FUNCTION_BLOCK EM_Doors EXTENDS EM_Base
VAR CONSTANT 
	c_nResultDataSize : UINT := 20;
END_VAR
VAR
//------------------------------------------//
//Control Modules (Devices)
	s_cmSpeedDoorOuter : CM_SpeedDoor;
	s_cmDoorLockCleanroom : CM_DoorLock;
//------------------------------------------//

//------------------------------------------//
//Inputs
	s_diTableDownSensor	: FB_DigInput;
	s_diBtnTableDown	: FB_DigInput;
	s_diBtnStop			: FB_DigInput;
	
//------------------------------------------//
	s_doRelayTableDown : FB_DigOutput;
//------------------------------------------//
//Outputs

//------------------------------------------//

//------------------------------------------//
//Params
	//Tool settings
	s_fbParamToolHardwareNr				: FB_HmiParamHandler;
    s_fbParamToolSoftwareVersion		: FB_HmiParamHandler;

	s_fbParamName						: FB_HmiParamHandler;
	s_fbParamNumber						: FB_HmiParamHandler;
	s_fbParamRevision                   : FB_HmiParamHandler;
	
	s_fbParamTeslaMeterIp				: FB_HmiParamHandler;
	s_fbParamTeslaMeterPort				: FB_HmiParamHandler;
	
	//Product settings (Maybe)
	s_fbParamTotalStroke				: FB_HmiParamHandler;
	s_fbParamStepStroke					: FB_HmiParamHandler;
	s_fbParamAveragingNumberTest		: FB_HmiParamHandler;
	
	s_fbParamaMaxMagnitudeCriteria		: FB_HmiParamHandler;
	
	s_fbParamRefIduBottom				: FB_HmiParamHandler;
	s_fbParamRefItm                     : FB_HmiParamHandler;
	s_fbParamRefCenterTpmPipe           : FB_HmiParamHandler;
	s_fbParamRefCpValve					: FB_HmiParamHandler;
//------------------------------------------//

//------------------------------------------//
//Variables
	s_sTestResult 						: STRING;
	
	s_eCurrentTest						: E_TestMode;
	s_stCommandsTesla					: ST_SCPI_TeslaCommands;
//------------------------------------------//

//------------------------------------------//
//Sensor data	
	s_aMagneticX						: ARRAY[0..c_nResultDataSize] OF LREAL;
	s_aMagneticY						: ARRAY[0..c_nResultDataSize] OF LREAL;
	s_aMagneticZ						: ARRAY[0..c_nResultDataSize] OF LREAL;
	s_aMagneticMagnitude				: ARRAY[0..c_nResultDataSize] OF LREAL;
	s_aProbePositionZ					: ARRAY[0..c_nResultDataSize] OF LREAL;
	
	s_sXMLData							: STRING(Param_Project.n_MaxLenghtXmlDbRow*Param_Project.n_NumberofRowsXmlDb);
	
	s_aHmi_MagneticTest					: ARRAY[1..3,0..c_nResultDataSize] OF ST_POINT;
	
//	s_aHmi_ProbePositionZ				: ARRAY[1..1,1..GVL_Datalogging.c_nHmiLogSize] OF ST_POINT;
//------------------------------------------//

//------------------------------------------//
//Alarms

//------------------------------------------//

//------------------------------------------//
//Hmi
	s_nToHmiStepNr						: INT;
	s_nToHmiMaxStepNr					: INT;
	s_sToHmiInstructionText				: T_MAXSTRING;
	s_sToHmiProcedure					: T_MAXSTRING;
	
	s_fbHmiBtnStart						: FB_HmiBtn;
	s_fbHmiBtnStop						: FB_HmiBtn;	
	s_fbHmiBtnDiagnosticsLogging		: FB_HmiBtn;
	
	s_fbHmiProbeMotor 					: Hmi_Motor_Base;
	
	s_fbHmiBtnEnableMotor				: FB_HmiBtn;
	s_fbHmiBtnHomeMotor					: FB_HmiBtn;
	s_fbHmiBtnGetField					: FB_HmiBtn;
	
	s_fbHmiLedHomedMotor				: FB_HmiLed;
	s_fbHmiTableDownPressed				: FB_HmiLed;
	s_fbHmiStopPressed					: FB_HmiLed;
	s_fbHmiTableDownSensor				: FB_HmiLed;
//------------------------------------------//
END_VAR


SUPER^();

METHOD Protected _m_Alarms : BOOL
IF NOT SUPER^._m_Alarms() THEN
	RETURN;
END_IF

_m_Alarms := TRUE;
END_METHOD

METHOD PRIVATE _m_DatabaseMagnetic : BOOL
VAR_INPUT
	i_bCmdReset						: BOOL;
	i_sPassFail						: STRING;
END_VAR
VAR_INST
	s_aDbColumns				: ARRAY[1..GVL_DataLogging.c_nDbColumnMagnetic] OF STRING;
	s_aDbColumnValues			: ARRAY[1..GVL_DataLogging.c_nDbColumnMagnetic] OF STRING;
	
	s_nCounterDbLogging				: UINT := 1;
END_VAR
IF i_bCmdReset THEN
	s_nCounterDbLogging 	:= 1;
	
	MEMSET(ADR(s_aDbColumns), 0 , SIZEOF(s_aDbColumns));
	MEMSET(ADR(s_aDbColumnValues), 0 , SIZEOF(s_aDbColumnValues));	

	s_aDbColumns[1] 		:= 'TestTool Hardware Nr';
	s_aDbColumns[2] 		:= 'TestTool Software Version';
	s_aDbColumns[3] 		:= 'User';
	s_aDbColumns[4] 		:= 'Serial number';
	s_aDbColumns[5] 		:= '12NC';
	s_aDbColumns[6] 		:= 'Notes';
	s_aDbColumns[7] 		:= 'PassFail';
	s_aDbColumns[8] 		:= 'Message';
	s_aDbColumns[9] 		:= 'Measurement';
	
	s_aDbColumnValues[1] 	:= GVL_DataLogging.g_stReportData.CabinetSerialNumber;
	s_aDbColumnValues[2] 	:= GVL_DataLogging.g_stReportData.TesterSoftwareVersion;
	s_aDbColumnValues[3] 	:= GVL.g_sUser;
	s_aDbColumnValues[4] 	:= GVL_DataLogging.g_stReportData.SerialNumber;;
	s_aDbColumnValues[5] 	:= CONCAT(s_fbParamNumber.p_sValue, CONCAT('^' ,TO_STRING(TO_INT(s_fbParamRevision.p_fValue))));
	s_aDbColumnValues[6] 	:= GVL.g_sNotesEntry;
	s_aDbColumnValues[7]  	:= i_sPassFail;
		
	IF GVL_KMWEGenericLib.g_fbAlarmManager.p_bAlarmActive THEN
		s_aDbColumnValues[8] 	:= 'Stopped due to Alarm';
	ELSE
		s_aDbColumnValues[8] 	:= '';
	END_IF
	
END_IF

IF s_nCounterDbLogging < GVL_DataLogging.c_nDbColumnMagnetic THEN
	IF GVL_Datalogging.g_fbSqlDatabase.m_UpdateTableValue(i_sTableName					:= GVL_DataLogging.c_sTableNameMagnetic,
															i_sIdentificationColumnName := GVL_DataLogging.c_sIdentificationColumnDataTime,
															i_sIdentificationValue		:= GVL_KMWEGenericLib.g_fbCurrentTime.p_sCurrentDateTime_DB, 
															i_sColumnName				:= s_aDbColumns[s_nCounterDbLogging], 
															i_sColumnValue				:= s_aDbColumnValues[s_nCounterDbLogging])
	THEN
		IF s_nCounterDbLogging <=  GVL_DataLogging.c_nDbColumnMagnetic THEN
			s_nCounterDbLogging := s_nCounterDbLogging + 1;
		END_IF
	END_IF
ELSIF s_nCounterDbLogging = GVL_DataLogging.c_nDbColumnMagnetic THEN
	IF GVL_Datalogging.g_fbSqlDatabase.m_UpdateTableXml(i_sTableName					:= GVL_DataLogging.c_sTableNameMagnetic,
															i_sIdentificationColumnName := GVL_DataLogging.c_sIdentificationColumnDataTime,
															i_sIdentificationValue		:= GVL_KMWEGenericLib.g_fbCurrentTime.p_sCurrentDateTime_DB, 
															i_sColumnName				:= s_aDbColumns[s_nCounterDbLogging], 
															i_addrColumnValue			:= ADR(s_sXMLData))
	THEN
		IF s_nCounterDbLogging <=  GVL_DataLogging.c_nDbColumnMagnetic THEN
			s_nCounterDbLogging := s_nCounterDbLogging + 1;
		END_IF
	END_IF
END_IF

_m_DatabaseMagnetic := s_nCounterDbLogging > GVL_DataLogging.c_nDbColumnMagnetic;
END_METHOD

METHOD Protected _m_Devices : BOOL
VAR_INPUT
END_VAR
IF NOT SUPER^._m_Devices() THEN
	RETURN;
END_IF

s_CmProbeMotor(
	i_bReqEnable					:= , //written in test procedure or manual 
	i_eCtrlMode						:= i_eCtrlMode, 
	i_bCmdReset						:= i_bCmdReset, 
	i_sCmName						:= 'Probe motor');	
	
s_CmTeslaMeter(
	i_bReqEnable					:= , //written in test procedure or manual  
	i_eCtrlMode						:= i_eCtrlMode, 
	i_bCmdReset						:= i_bCmdReset, 
	i_sCmName						:= 'Tesla meter');
	
_m_Devices := TRUE;
END_METHOD

METHOD PRIVATE _m_GetMagneticField : E_STATE
VAR_INPUT
	i_bCmdReset			: BOOL;
END_VAR
VAR_OUTPUT
	q_fMagneticX		: LREAL;
	q_fMagneticY		: LREAL;
	q_fMagneticZ		: LREAL;
END_VAR
VAR_INST
	//Sequence control
	s_eSequence				: E_ModuleSeqBase;
	s_fbSeqControl			: FB_SeqControl;
	
	s_nInternalStep			: UINT := 0;
	
	//Communication
	s_aReplyBuffer			: ARRAY[1..100] OF T_MAXSTRING; //Tesla
	s_aResults				: ARRAY[1..10 ] OF T_MAXSTRING;	//Tesla
	s_sReply				: T_MAXSTRING;
	s_nIndexReply 			: UDINT := 1;
	s_nIndexResults			: UDINT := 1;
	
	t_nMeasurementsReceived		: UDINT := 1;

	//Measurements
	s_aMagneticXAve			: ARRAY[1..100] OF LREAL;
	s_aMagneticYAve			: ARRAY[1..100] OF LREAL;
	s_aMagneticZAve			: ARRAY[1..100] OF LREAL;
END_VAR
VAR
	t_nCyclceReplies			: UDINT := 1;
	
	t_fAveragingX				: LREAL;
	t_fAveragingY				: LREAL;
	t_fAveragingZ				: LREAL;

END_VAR
s_fbSeqControl(
	i_nSeqStep:= s_eSequence, 
	i_sStepName:= TO_STRING(s_eSequence), 
	i_bCmdReset:= i_bCmdReset, 
	i_bStaError:= FALSE,  
	q_eActState=> _m_GetMagneticField);
	
CASE s_eSequence OF
	E_ModuleSeqBase.Idle:
		;
		
	E_ModuleSeqBase.Start:
		IF s_fbSeqControl.q_bStaEntry THEN
			s_nInternalStep := s_nInternalStep + 1;
		END_IF
		
		IF s_fbSeqControl.q_tmStepTime > T#2S OR s_nInternalStep > 1 THEN
			IF s_CmTeslaMeter.m_SendCommand(i_sCommand := s_stCommandsTesla.sGetMeasurents , i_bAddCRChar := TRUE) THEN
				s_eSequence 	:= E_ModuleSeqBase.Busy;
			END_IF
		END_IF

	E_ModuleSeqBase.Busy:
		IF s_fbSeqControl.q_bStaEntry THEN
			t_nMeasurementsReceived := 1;
		END_IF
		
		s_CmTeslaMeter.m_ReadReplyBuffer(q_sReply => s_sReply);
			
		IF s_sReply <> 'No reply' THEN
			IF t_nMeasurementsReceived = 1 THEN
				s_aReplyBuffer[t_nCyclceReplies] := '';
				t_nMeasurementsReceived := 2;
			ELSIF t_nMeasurementsReceived = 2 THEN
				s_aMagneticXAve[s_nInternalStep] := TO_LREAL(s_aReplyBuffer[t_nCyclceReplies]);
				s_aMagneticXAve[s_nInternalStep] := TO_LREAL(s_sReply);
				s_aReplyBuffer[t_nCyclceReplies] := '';
				t_nMeasurementsReceived := 3;
			ELSIF t_nMeasurementsReceived = 3 THEN
				s_aMagneticYAve[s_nInternalStep] := TO_LREAL(s_aReplyBuffer[t_nCyclceReplies]);
				s_aMagneticYAve[s_nInternalStep] := TO_LREAL(s_sReply);
				s_aReplyBuffer[t_nCyclceReplies] := '';
				t_nMeasurementsReceived := 4;
			ELSIF t_nMeasurementsReceived = 4 THEN
				s_aMagneticZAve[s_nInternalStep] := TO_LREAL(s_aReplyBuffer[t_nCyclceReplies]);
				s_aMagneticZAve[s_nInternalStep] := TO_LREAL(s_sReply);
				s_aReplyBuffer[t_nCyclceReplies] := '';

				IF s_nInternalStep = TO_UINT(s_fbParamAveragingNumberTest.p_fValue) THEN
					s_eSequence := E_ModuleSeqBase.Ready;
				ELSE
					s_eSequence := E_ModuleSeqBase.Start;
				END_IF 
			END_IF
		END_IF

	E_ModuleSeqBase.Ready:
		IF s_fbSeqControl.q_bStaEntry THEN
			s_nInternalStep := 0;
			
			t_fAveragingX	:= 0;
			t_fAveragingY	:= 0;
			t_fAveragingZ	:= 0;
 
			MEMSET(ADR(s_aReplyBuffer)			, 0, SIZEOF(s_aReplyBuffer));
			MEMSET(ADR(s_aResults)				, 0, SIZEOF(s_aResults));
		END_IF
		
		FOR t_nCyclceReplies := 1 TO 100 DO
			t_fAveragingX := t_fAveragingX + s_aMagneticXAve[t_nCyclceReplies];
			t_fAveragingY := t_fAveragingY + s_aMagneticYAve[t_nCyclceReplies];
			t_fAveragingZ := t_fAveragingZ + s_aMagneticZAve[t_nCyclceReplies];

			IF t_nCyclceReplies = 100 THEN
			MEMSET(ADR(s_aMagneticXAve)			, 0, SIZEOF(s_aMagneticXAve));
			MEMSET(ADR(s_aMagneticYAve)			, 0, SIZEOF(s_aMagneticYAve));
			MEMSET(ADR(s_aMagneticZAve)			, 0, SIZEOF(s_aMagneticZAve));				
			END_IF
		END_FOR
			
			q_fMagneticX	:= t_fAveragingX/s_fbParamAveragingNumberTest.p_fValue;
			q_fMagneticY	:= t_fAveragingY/s_fbParamAveragingNumberTest.p_fValue;
			q_fMagneticZ	:= t_fAveragingZ/s_fbParamAveragingNumberTest.p_fValue;
				
	E_ModuleSeqBase.Error:
		;
END_CASE
END_METHOD

METHOD Protected _m_Hmi : BOOL
VAR_INPUT
END_VAR
VAR_INST
END_VAR
IF NOT SUPER^._m_Hmi() THEN
	RETURN;
END_IF

s_fbHmiBtnDiagnosticsLogging();
s_fbHmiBtnStart();
s_fbHmiBtnStop();

s_fbHmiBtnEnableMotor();
s_fbHmiBtnHomeMotor();
s_fbHmiBtnGetField();

s_fbHmiProbeMotor(i_IMotor := s_CmProbeMotor);

s_fbHmiLedHomedMotor(i_bStaLed := s_CmProbeMotor.p_bStaMotorHomed);
s_fbHmiTableDownPressed(i_bStaLed := s_diBtnTableDown.p_bStaInput);
s_fbHmiTableDownSensor(i_bStaLed := s_diTableDownSensor.p_bStaInput);
s_fbHmiStopPressed(i_bStaLed := s_diBtnStop.p_bStaInput);

_m_Hmi := TRUE;
END_METHOD

METHOD PRIVATE _m_HmiPlots
VAR CONSTANT 

END_VAR
VAR_INPUT
	i_bStaHmiLogging : BOOL;
END_VAR
VAR_INST
	s_tonDiagnosticsHmi 	: TON;	

	s_osrDiagnositcsHmi		: R_TRIG;
	s_osfDiagnositcsHmi		: F_TRIG;
	
	s_nInternalTestTime		: LREAL;
	
	s_nCounterDiagRawArray	: UDINT;
	
	s_nCounterPolish		: UDINT;
	
	s_fStartVolumePumped 	: LREAL;
END_VAR
s_tonDiagnosticsHmi(IN := NOT s_tonDiagnosticsHmi.Q, PT := TO_TIME(1000/c_tmHmiLogFreq));

s_osrDiagnositcsHmi(CLK := i_bStaHmiLogging);
s_osfDiagnositcsHmi(CLK := i_bStaHmiLogging);

IF s_osrDiagnositcsHmi.Q THEN
	s_nCounterDiagRawArray 	:= 1;
	
	s_fStartVolumePumped	:= s_fPumpedVolume;
	
	MEMSET(ADR(s_aHmiMovingAve_WaterPresure), 0, SIZEOF(s_aHmiMovingAve_WaterPresure));
	MEMSET(ADR(s_aHmiMovingAve_R14Pressure), 0, SIZEOF(s_aHmiMovingAve_R14Pressure));
	MEMSET(ADR(s_aHmiMovingAve_WaterTemperature), 0, SIZEOF(s_aHmiMovingAve_WaterTemperature));
	MEMSET(ADR(s_aHmiMovingAve_R14Temperature), 0, SIZEOF(s_aHmiMovingAve_R14Temperature));
	MEMSET(ADR(s_aHmi_PumpedWaterVolume), 0, SIZEOF(s_aHmi_PumpedWaterVolume));
	MEMSET(ADR(s_aHmi_VoltageMeasurement), 0, SIZEOF(s_aHmi_VoltageMeasurement));
	MEMSET(ADR(s_aHmi_MovingAve_TemperatureCombined), 0, SIZEOF(s_aHmi_MovingAve_TemperatureCombined));
	MEMSET(ADR(s_aHmi_MovingAve_PressureCombined), 0, SIZEOF(s_aHmi_MovingAve_PressureCombined));
	
END_IF

IF i_bStaHmiLogging AND s_tonDiagnosticsHmi.Q THEN
	
		FOR s_nCounterPolish := s_nCounterDiagRawArray TO c_nHmiLogSize DO
			IF s_nCounterDiagRawArray > 1 THEN
				s_aHmiMovingAve_WaterPresure[1,s_nCounterPolish].x 		:= s_aHmiMovingAve_WaterPresure[1,s_nCounterDiagRawArray-1].x;
				s_aHmiMovingAve_R14Pressure[1,s_nCounterPolish].x 		:= s_aHmiMovingAve_R14Pressure[1,s_nCounterDiagRawArray-1].x;
				s_aHmiMovingAve_WaterTemperature[1,s_nCounterPolish].x 	:= s_aHmiMovingAve_WaterTemperature[1,s_nCounterDiagRawArray-1].x;
				s_aHmiMovingAve_R14Temperature[1,s_nCounterPolish].x 	:= s_aHmiMovingAve_R14Temperature[1,s_nCounterDiagRawArray-1].x;
				s_aHmi_PumpedWaterVolume[1,s_nCounterPolish].x			:= s_aHmi_PumpedWaterVolume[1,s_nCounterDiagRawArray-1].x;
				s_aHmi_VoltageMeasurement[1,s_nCounterPolish].x			:= s_aHmi_VoltageMeasurement[1,s_nCounterDiagRawArray-1].x;
				
				s_aHmi_MovingAve_TemperatureCombined[1,s_nCounterPolish].x 	:= s_aHmi_MovingAve_TemperatureCombined[1,s_nCounterDiagRawArray-1].x;		
				s_aHmi_MovingAve_TemperatureCombined[2,s_nCounterPolish].x 	:= s_aHmi_MovingAve_TemperatureCombined[2,s_nCounterDiagRawArray-1].x;
				s_aHmi_MovingAve_PressureCombined[1,s_nCounterPolish].x 	:= s_aHmi_MovingAve_PressureCombined[1,s_nCounterDiagRawArray-1].x;		
				s_aHmi_MovingAve_PressureCombined[2,s_nCounterPolish].x 	:= s_aHmi_MovingAve_PressureCombined[2,s_nCounterDiagRawArray-1].x;
		
				s_aHmiMovingAve_WaterPresure[1,s_nCounterPolish].y 		:= s_aHmiMovingAve_WaterPresure[1,s_nCounterDiagRawArray-1].y;
				s_aHmiMovingAve_R14Pressure[1,s_nCounterPolish].y		:= s_aHmiMovingAve_R14Pressure[1,s_nCounterDiagRawArray-1].y;
				s_aHmiMovingAve_WaterTemperature[1,s_nCounterPolish].y 	:= s_aHmiMovingAve_WaterTemperature[1,s_nCounterDiagRawArray-1].y;
				s_aHmiMovingAve_R14Temperature[1,s_nCounterPolish].y 	:= s_aHmiMovingAve_R14Temperature[1,s_nCounterDiagRawArray-1].y;
				s_aHmi_PumpedWaterVolume[1,s_nCounterPolish].y 			:= s_aHmi_PumpedWaterVolume[1,s_nCounterDiagRawArray-1].y;
				s_aHmi_VoltageMeasurement[1,s_nCounterPolish].y 		:= s_aHmi_VoltageMeasurement[1,s_nCounterDiagRawArray-1].y;
				
				s_aHmi_MovingAve_TemperatureCombined[1,s_nCounterPolish].y 	:= s_aHmi_MovingAve_TemperatureCombined[1,s_nCounterDiagRawArray-1].y;		
				s_aHmi_MovingAve_TemperatureCombined[2,s_nCounterPolish].y 	:= s_aHmi_MovingAve_TemperatureCombined[2,s_nCounterDiagRawArray-1].y;
				s_aHmi_MovingAve_PressureCombined[1,s_nCounterPolish].y 	:= s_aHmi_MovingAve_PressureCombined[1,s_nCounterDiagRawArray-1].y;		
				s_aHmi_MovingAve_PressureCombined[2,s_nCounterPolish].y 	:= s_aHmi_MovingAve_PressureCombined[2,s_nCounterDiagRawArray-1].y;
			END_IF
		END_FOR
		
	//Raw data logging of sensor (Discuss with marco if this can be raw or needs to be the low pass filter data)
	IF s_nCounterDiagRawArray <= c_nHmiLogSize THEN
		s_aHmiMovingAve_WaterPresure[1,s_nCounterDiagRawArray].x 		   	:= (TO_LREAL(s_nCounterDiagRawArray)*(1/TO_LREAL(c_tmHmiLogFreq)));
		s_aHmiMovingAve_R14Pressure[1,s_nCounterDiagRawArray].x 		    := (TO_LREAL(s_nCounterDiagRawArray)*(1/TO_LREAL(c_tmHmiLogFreq)));
		s_aHmiMovingAve_WaterTemperature[1,s_nCounterDiagRawArray].x 		:= (TO_LREAL(s_nCounterDiagRawArray)*(1/TO_LREAL(c_tmHmiLogFreq)));
		s_aHmiMovingAve_R14Temperature[1,s_nCounterDiagRawArray].x 	  		:= (TO_LREAL(s_nCounterDiagRawArray)*(1/TO_LREAL(c_tmHmiLogFreq)));
		s_aHmi_PumpedWaterVolume[1,s_nCounterDiagRawArray].x			    := (TO_LREAL(s_nCounterDiagRawArray)*(1/TO_LREAL(c_tmHmiLogFreq)));
		s_aHmi_VoltageMeasurement[1,s_nCounterDiagRawArray].x			    := (TO_LREAL(s_nCounterDiagRawArray)*(1/TO_LREAL(c_tmHmiLogFreq)));
		s_aHmi_MovingAve_TemperatureCombined[1,s_nCounterDiagRawArray].x 	:= (TO_LREAL(s_nCounterDiagRawArray)*(1/TO_LREAL(c_tmHmiLogFreq)));
		s_aHmi_MovingAve_TemperatureCombined[2,s_nCounterDiagRawArray].x 	:=(TO_LREAL(s_nCounterDiagRawArray)*(1/TO_LREAL(c_tmHmiLogFreq)));
		s_aHmi_MovingAve_PressureCombined[1,s_nCounterDiagRawArray].x 		:= (TO_LREAL(s_nCounterDiagRawArray)*(1/TO_LREAL(c_tmHmiLogFreq)));
		s_aHmi_MovingAve_PressureCombined[2,s_nCounterDiagRawArray].x 		:=(TO_LREAL(s_nCounterDiagRawArray)*(1/TO_LREAL(c_tmHmiLogFreq)));

		s_aHmiMovingAve_WaterPresure[1,s_nCounterDiagRawArray].y			:= s_fbMvAveWaterPressure.p_fMovingAverage;       
		s_aHmiMovingAve_R14Pressure[1,s_nCounterDiagRawArray].y				:= s_fbMvAveR14Pressure.p_fMovingAverage;  
		s_aHmiMovingAve_WaterTemperature[1,s_nCounterDiagRawArray].y		:= s_fbMvAveWaterTemperature.p_fMovingAverage;      
		s_aHmiMovingAve_R14Temperature[1,s_nCounterDiagRawArray].y			:= s_fbMvAveR14Temperature.p_fMovingAverage;
		s_aHmi_PumpedWaterVolume[1,s_nCounterDiagRawArray].y				:= s_fPumpedVolume - s_fStartVolumePumped;
		s_aHmi_VoltageMeasurement[1,s_nCounterDiagRawArray].y				:=  s_CmVoltageMeasurement.p_fMeasurement;
	
		s_aHmi_MovingAve_TemperatureCombined[1,s_nCounterDiagRawArray].y 	:= s_fbMvAveWaterTemperature.p_fMovingAverage;  
		s_aHmi_MovingAve_TemperatureCombined[2,s_nCounterDiagRawArray].y 	:= s_fbMvAveR14Temperature.p_fMovingAverage;
		s_aHmi_MovingAve_PressureCombined[1,s_nCounterDiagRawArray].y 		:= s_fbMvAveWaterPressure.p_fMovingAverage;     
		s_aHmi_MovingAve_PressureCombined[2,s_nCounterDiagRawArray].y 		:= s_fbMvAveR14Pressure.p_fMovingAverage;  

	END_IF
	
	s_nCounterDiagRawArray := s_nCounterDiagRawArray + 1;

END_IF
END_METHOD

METHOD PRIVATE _m_HmiPlots_Test
VAR_INPUT
	i_bStaHmiLogging 	: BOOL;
	i_bNewMeasurement	: BOOL;
END_VAR
VAR_INST
	s_tonDiagnosticsHmi 	: TON;	

	s_osrDiagnositcsHmi		: R_TRIG;
	s_osfDiagnositcsHmi		: F_TRIG;
	
	s_osrDiagnositcsHmi		: R_TRIG;
	s_osfDiagnositcsHmi		: F_TRIG;
	
	s_nCounterMeasurements	: UDINT;
	
	s_nCounterPolish		: UDINT;
	
	s_fStartVolumePumped 	: LREAL;
END_VAR
s_osrDiagnositcsHmi(CLK := i_bStaHmiLogging);
s_osfDiagnositcsHmi(CLK := i_bStaHmiLogging);

IF s_osrDiagnositcsHmi.Q THEN
	s_nCounterMeasurements 	:= 1;
		
	MEMSET(ADR(s_aHmi_MagneticTest), 0, SIZEOF(s_aHmi_MagneticTest));
END_IF

IF i_bStaHmiLogging AND i_bNewMeasurement THEN
	FOR s_nCounterPolish := s_nCounterMeasurements TO c_nResultDataSize DO
		IF s_nCounterMeasurements > 1 THEN
			s_aHmi_MagneticTest[1,s_nCounterPolish].x 			:= s_aHmi_MagneticTest[1,s_nCounterMeasurements-1].x;
			s_aHmi_MagneticTest[2,s_nCounterPolish].x 			:= s_aHmi_MagneticTest[2,s_nCounterMeasurements-1].x;
			s_aHmi_MagneticTest[3,s_nCounterPolish].x 			:= s_aHmi_MagneticTest[3,s_nCounterMeasurements-1].x;
			s_aHmi_MagneticTest[4,s_nCounterPolish].x 			:= s_aHmi_MagneticTest[4,s_nCounterMeasurements-1].x;

			s_aHmi_MagneticTest[1,s_nCounterPolish].y			:= s_aHmi_MagneticTest[1,s_nCounterMeasurements-1].y;
			s_aHmi_MagneticTest[2,s_nCounterPolish].y			:= s_aHmi_MagneticTest[2,s_nCounterMeasurements-1].y;
			s_aHmi_MagneticTest[3,s_nCounterPolish].y			:= s_aHmi_MagneticTest[3,s_nCounterMeasurements-1].y;
			s_aHmi_MagneticTest[4,s_nCounterPolish].y 			:= s_aHmi_MagneticTest[4,s_nCounterMeasurements-1].y;
		END_IF
	END_FOR
	
	s_nCounterMeasurements := s_nCounterMeasurements + 
END_IF
END_METHOD

METHOD Protected _m_Init : BOOL
VAR_INPUT
END_VAR
IF NOT SUPER^._m_Init() THEN
	RETURN;
END_IF

//----------------------------------//
//CM
	s_CmProbeMotor.i_bReqEnable						:= FALSE;
	s_CmProbeMotor.i_sCmName 						:= 'Probe motor';
	s_CmProbeMotor.i_eBtnCtrlType					:= E_HmiButtonType.PUSHBUTTON;
	s_CmProbeMotor.i_bCfgReverseDirection			:= FALSE;
	s_CmProbeMotor.p_bCfgMovingForward				:= TRUE;
	s_CmProbeMotor.p_bCfgMovingReverse				:= TRUE;
	s_CmProbeMotor.p_fSetMotorVelo					:= 10;
	
	s_CmProbeMotor.i_stSettings.i_fAccelaration 	:= 1000;
	s_CmProbeMotor.i_stSettings.i_fDecelaration		:= 1000;
	s_CmProbeMotor.i_stSettings.i_fJerk				:= 10000;
	
	s_CmTeslaMeter.i_bReqEnable						:= FALSE;
	s_CmTeslaMeter.i_stSettings.tConnectionTimeOut	:= T#5S;

	
//---------------------------------//	
	
//----------------------------------//	
//Hmi 
	s_fbHmiBtnDiagnosticsLogging.p_eButtontype 			:= E_HmiButtonType.TOGGLEBUTTON;
	s_fbHmiBtnDiagnosticsLogging.p_bStaVisible 			:= TRUE;
	s_fbHmiBtnDiagnosticsLogging.p_bStaEnabled 			:= TRUE;
	s_fbHmiBtnDiagnosticsLogging.p_sBtnText				:= 'Diagnostics Logging';
	
	s_fbHmiBtnStart.p_eButtontype 						:= E_HmiButtonType.PUSHBUTTON;
	s_fbHmiBtnStart.p_bStaVisible 						:= FALSE;
	s_fbHmiBtnStart.p_bStaEnabled 						:= FALSE;		
	s_fbHmiBtnStart.p_sBtnText							:= 'Start';

	s_fbHmiBtnStop.p_eButtontype 						:= E_HmiButtonType.PUSHBUTTON;
	s_fbHmiBtnStop.p_bStaVisible 						:= FALSE;
	s_fbHmiBtnStop.p_bStaEnabled 						:= FALSE;		
	s_fbHmiBtnStop.p_sBtnText							:= 'Stop';
	
	s_fbHmiBtnEnableMotor.p_eButtontype 				:= E_HmiButtonType.TOGGLEBUTTON;
	s_fbHmiBtnEnableMotor.p_bStaVisible 				:= TRUE;
	s_fbHmiBtnEnableMotor.p_bStaEnabled 				:= FALSE;		
	s_fbHmiBtnEnableMotor.p_sBtnText					:= 'Enable motor';
	
	s_fbHmiBtnGetField.p_eButtontype 					:= E_HmiButtonType.PUSHBUTTON;
	s_fbHmiBtnGetField.p_bStaVisible 					:= TRUE;
	s_fbHmiBtnGetField.p_bStaEnabled 					:= FALSE;		
	s_fbHmiBtnGetField.p_sBtnText						:= 'Get magnetic field';
	
	s_fbHmiBtnHomeMotor.p_eButtontype 					:= E_HmiButtonType.PUSHBUTTON;
	s_fbHmiBtnHomeMotor.p_bStaVisible 					:= TRUE;
	s_fbHmiBtnHomeMotor.p_bStaEnabled 					:= FALSE;		
	s_fbHmiBtnHomeMotor.p_sBtnText						:= 'Home motor';
//----------------------------------//	


//----------------------------------//	
//Initialize all moving averages

//----------------------------------//	

//----------------------------------//	
//Inputs
s_diTableDownSensor.i_stSettings.tmInputDelay	:= T#0S;	
s_diBtnTableDown.i_stSettings.tmInputDelay		:= T#0S;
s_diBtnStop.i_stSettings.tmInputDelay			:= T#0S;
//----------------------------------//	

//----------------------------------//	
//Inputs
s_doRelayTableDown.i_stSettings.bCfgDelay		:= FALSE;	
s_doRelayTableDown.i_stSettings.tmOutputDelay	:= T#0S;	
//----------------------------------//	

_m_Init := TRUE;
END_METHOD

METHOD PROTECTED _m_Inputs : BOOL
VAR_INPUT
END_VAR
IF NOT SUPER^._m_Inputs() THEN
	RETURN;
END_IF

s_diTableDownSensor();
s_diBtnTableDown();	
s_diBtnStop();			

_m_Inputs := TRUE;
END_METHOD

METHOD PRIVATE _m_Manual : E_STATE
VAR_INPUT
	i_bCmdReset			: BOOL;
	i_bStaError			: BOOL;
END_VAR
VAR_INST
	//Sequence control
	s_eSequence				: E_ManualMode_Steps;
	s_fbSeqControl			: FB_SeqControl;
	
	s_nInternalStep			: UINT := 0;
	
	//Communication
	s_aReplyBuffer			: ARRAY[1..100] OF T_MAXSTRING; //Tesla
	s_aResults				: ARRAY[1..10 ] OF T_MAXSTRING;	//Tesla
	s_sReply				: T_MAXSTRING;
	s_nIndexReply 			: UDINT := 1;
	s_nIndexResults			: UDINT := 1;
	
	//Measurements
	s_fMagneticX			: LREAL;
	s_fMagneticY			: LREAL;
	s_fMagneticZ			: LREAL;
	s_fMagneticMagnitude 	: LREAL;
END_VAR
VAR
	t_nCyclceReplies			: UDINT := 1;
	t_nMeasurementsReceived		: UDINT := 1;
	
	t_fAveragingX				: LREAL;
	t_fAveragingY				: LREAL;
	t_fAveragingZ				: LREAL;

END_VAR
s_fbSeqControl(
	i_nSeqStep:= s_eSequence, 
	i_sStepName:= TO_STRING(s_eSequence), 
	i_bCmdReset:= i_bCmdReset, 
	i_bStaError:= i_bStaError,  
	q_eActState=> _m_Manual);
	
IF GVL_KMWEGenericLib.g_fbHmiBtnReturn.p_osrBtnPress AND s_eSequence <> E_ManualMode_Steps.Error AND s_eSequence <> E_ManualMode_Steps.Start THEN
	s_eSequence := E_ManualMode_Steps.Error;
END_IF

IF GVL.g_sToHmiMiddleContent = GVL.g_stHmiMiddle.AlarmManager THEN
	GVL_KMWEGenericLib.g_fbHmiBtnReturn.p_sBtnText	 	:= 'Return';
END_IF

CASE s_eSequence OF
	E_ManualMode_Steps.Idle:
		;
		
	E_ManualMode_Steps.Start:
		IF s_fbSeqControl.q_bStaEntry THEN
			GVL.g_eStaLedColor := E_KmweLedColors.Green;
			
			s_fbHmiBtnEnableMotor.p_bStaEnabled 						:= TRUE;
			s_fbHmiBtnGetField.p_bStaEnabled 							:= TRUE;
			GVL_KMWEGenericLib.g_fbHmiBtnReturnToStart.p_bStaEnabled 	:= TRUE;
		END_IF
	
		IF GVL.g_sToHmiMiddleContent <> GVL.g_stHmiMiddle.AlarmManager THEN
			GVL_KMWEGenericLib.g_fbHmiBtnReturn.p_bStaEnabled 	:= FALSE;
			GVL_KMWEGenericLib.g_fbHmiBtnReturn.p_bStaVisible 	:= FALSE;
			GVL_KMWEGenericLib.g_fbHmiBtnReturn.p_sBtnText	 	:= 'Return';
		END_IF
		
		IF s_fbHmiBtnEnableMotor.p_osrBtnPress OR s_fbHmiBtnEnableMotor.p_osfBtnPress THEN
			GVL_KMWEGenericLib.g_fbHmiBtnReturn.p_bStaEnabled 	:= TRUE;
			GVL_KMWEGenericLib.g_fbHmiBtnReturn.p_bStaVisible 	:= TRUE;
			GVL_KMWEGenericLib.g_fbHmiBtnReturn.p_sBtnText	 	:= 'Stop action';		
		
			s_fbHmiBtnEnableMotor.p_bStaEnabled 						:= FALSE;
			s_fbHmiBtnHomeMotor.p_bStaEnabled							:= FALSE;
			s_fbHmiBtnGetField.p_bStaEnabled 							:= FALSE;
			
			GVL_KMWEGenericLib.g_fbHmiBtnReturnToStart.p_bStaEnabled 	:= FALSE;
			s_eSequence 												:= E_ManualMode_Steps.EnableDisableMotor;
		END_IF
		
		IF s_fbHmiBtnGetField.p_osrBtnPress THEN
			GVL_KMWEGenericLib.g_fbHmiBtnReturn.p_bStaEnabled 			:= TRUE;
			GVL_KMWEGenericLib.g_fbHmiBtnReturn.p_bStaVisible 			:= TRUE;
			GVL_KMWEGenericLib.g_fbHmiBtnReturn.p_sBtnText	 			:= 'Stop action';	
		                                                                
			GVL_KMWEGenericLib.g_fbHmiBtnReturnToStart.p_bStaEnabled 	:= FALSE;
			s_fbHmiBtnGetField.p_bStaEnabled 							:= FALSE;
			s_fbHmiBtnEnableMotor.p_bStaEnabled 						:= FALSE;
			
			s_fMagneticMagnitude										:= 0;
			                                                            
			s_eSequence													:= E_ManualMode_Steps.ConnectTesla;
		END_IF
		
		IF s_CmProbeMotor.p_bStaEnabled THEN
			IF s_fbHmiBtnHomeMotor.p_osrBtnPress THEN
				GVL_KMWEGenericLib.g_fbHmiBtnReturnToStart.p_bStaEnabled 	:= FALSE;
				s_eSequence 												:= E_ManualMode_Steps.HomeMotor;
			END_IF
		END_IF
		
		s_doRelayTableDown.i_bStaOutput	:= NOT s_diTableDownSensor.p_bStaInput 
											AND s_diBtnTableDown.p_bStaInput 
											AND NOT s_diBtnStop.p_bStaInput;
		
	E_ManualMode_Steps.EnableDisableMotor:
		IF s_fbHmiBtnEnableMotor.p_bStaBtn THEN
			s_CmProbeMotor.i_bReqEnable 			:= TRUE;
			s_CmProbeMotor.p_fSetMotorVelo			:= 100;
			
			IF s_CmProbeMotor.m_EnableAxis() THEN
				s_fbHmiBtnHomeMotor.p_bStaEnabled 	:= TRUE;
				s_eSequence 						:= E_ManualMode_Steps.Start;	
			END_IF
		END_IF
		
		IF NOT s_fbHmiBtnEnableMotor.p_bStaBtn THEN
			IF s_CmProbeMotor.m_DisableAxis() THEN
				s_fbHmiBtnHomeMotor.p_bStaEnabled 	:= FALSE;
				s_CmProbeMotor.i_bReqEnable 		:= FALSE;
				s_eSequence 						:= E_ManualMode_Steps.Start;	
			END_IF
		END_IF
		
	E_ManualMode_Steps.HomeMotor:
		IF s_fbSeqControl.q_bStaEntry THEN
			s_sToHmiInstructionText := 'Motor homing';	
		END_IF
		
		IF NOT GVL.g_fbHmiBtnSimulation.p_bStaBtn THEN
			IF s_CmProbeMotor.m_HomeMotor() OR (NOT s_CmProbeMotor.p_bStaHoming AND NOT s_fbSeqControl.q_bStaEntry) THEN
				s_eSequence := E_ManualMode_Steps.Start;
			END_IF
		ELSE
			IF s_CmProbeMotor.m_SetPosition(i_fPosition := 0) THEN
				s_eSequence := E_ManualMode_Steps.Start;
			END_IF
		END_IF

	E_ManualMode_Steps.ConnectTesla:
		IF s_fbSeqcontrol.q_bStaEntry THEN
			s_CmTeslaMeter.i_bReqEnable					:= TRUE;
			s_CmTeslaMeter.i_stSettings.sMetrelIpAdress := s_fbParamTeslaMeterIp.p_sValue;
			s_CmTeslaMeter.i_stSettings.sMetrelPort 	:= TO_UDINT(s_fbParamTeslaMeterPort.p_fValue);
		END_IF
		
		IF  s_CmTeslaMeter.m_Connect() THEN
			s_eSequence 	:= E_ManualMode_Steps.ConfigureTesla;
		END_IF
		
	E_ManualMode_Steps.ConfigureTesla:
		IF s_CmTeslaMeter.m_SendCommand(i_sCommand := s_stCommandsTesla.sSetModeDC , i_bAddCRChar := TRUE) THEN
			s_eSequence 	:= E_ManualMode_Steps.MeasureMagneticField;
		END_IF

	E_ManualMode_Steps.MeasureMagneticField:
		IF _m_GetMagneticField(i_bCmdReset 		:= s_fbSeqControl.q_bStaEntry,
								q_fMagneticX 	=> s_fMagneticX,
								q_fMagneticY 	=> s_fMagneticY,
								q_fMagneticZ 	=> s_fMagneticZ) = E_STATE.Ready 
		THEN
			s_fMagneticMagnitude := SQRT((s_fMagneticX*s_fMagneticX) + ((s_fMagneticY*s_fMagneticY)));

			s_eSequence := 	E_ManualMode_Steps.DisconnectTesla;
		END_IF
		
	E_ManualMode_Steps.DisconnectTesla:
		IF s_CmTeslaMeter.m_Disconnect() THEN
			s_CmTeslaMeter.i_bReqEnable					:= FALSE;
			s_eSequence 								:= E_ManualMode_Steps.Start;
		END_IF
	
	E_ManualMode_Steps.Error:
		IF s_fbSeqControl.q_bStaEntry THEN
			s_fbHmiBtnEnableMotor.m_Off();
			s_fbHmiBtnEnableMotor.p_bStaEnabled 	:= FALSE;
			s_fbHmiBtnHomeMotor.p_bStaEnabled	 	:= FALSE;
			
			GVL_KMWEGenericLib.g_fbHmiBtnReturnToStart.p_bStaVisible 	:= TRUE;
			GVL_KMWEGenericLib.g_fbHmiBtnReturnToStart.p_bStaEnabled 	:= TRUE;
		END_IF
		
		IF GVL.g_sToHmiMiddleContent <> GVL.g_stHmiMiddle.AlarmManager THEN
			GVL_KMWEGenericLib.g_fbHmiBtnReturn.p_bStaEnabled 	:= FALSE;
			GVL_KMWEGenericLib.g_fbHmiBtnReturn.p_bStaVisible 	:= FALSE;	
			GVL_KMWEGenericLib.g_fbHmiBtnReturn.p_sBtnText	 	:= 'Return';
		END_IF
	
		IF s_CmTeslaMeter.p_bConnected THEN
			IF s_CmTeslaMeter.m_Disconnect() THEN 
				s_CmTeslaMeter.i_bReqEnable := FALSE;
			END_IF
		ELSE
			s_CmTeslaMeter.i_bReqEnable := FALSE;
		END_IF
	
		IF s_CmProbeMotor.p_bStaMoving THEN
			s_CmProbeMotor.m_StopMoving();
		ELSIF s_CmProbeMotor.p_bStaEnabled THEN
			s_CmProbeMotor.m_DisableAxis();
		END_IF
		
		IF NOT GVL_KMWEGenericLib.g_fbAlarmManager.p_bAlarmActive AND NOT s_CmProbeMotor.p_bStaEnabled AND NOT s_CmTeslaMeter.p_bConnected THEN
			s_eSequence := E_ManualMode_Steps.Start;
		END_IF
END_CASE
END_METHOD

METHOD PROTECTED _m_Outputs : BOOL
VAR_INPUT
END_VAR
IF NOT SUPER^._m_Outputs() THEN
	RETURN;
END_IF

s_doRelayTableDown(); //i_bStaOutput written in procedure or manual mode

_m_Outputs := TRUE;
END_METHOD

METHOD PROTECTED _m_Params : BOOL
VAR_INST
	s_fToHmiXAxisMin	: LREAL;
	s_fToHmiXAxisMax	: LREAL;
	s_fToHmiYAxisMin	: LREAL;
	s_fToHmiYAxisMax	: LREAL;
END_VAR
IF NOT SUPER^._m_Params() THEN
	RETURN;
END_IF

s_fbParamToolHardwareNr(i_fDefaultValue				:= 0,
						i_nArrayFolderIndex			:= 1,
						i_sName						:= 'Harware ID',
						i_bIsNumber					:= FALSE);

s_fbParamToolSoftwareVersion(i_fDefaultValue		:= 0,
							i_nArrayFolderIndex		:= 1,
							i_sName					:= 'Software Version',
							i_bIsNumber				:= FALSE);

s_fbParamName(i_fDefaultValue						:= 0,
				i_nArrayFolderIndex					:= 1,
				i_sName								:= 'Description',
				i_bIsNumber							:= FALSE);
							
s_fbParamTeslaMeterIp(i_fDefaultValue			:= 0,
						i_nArrayFolderIndex		:= 1,
						i_sName					:= 'Tesla meter ip adress',
						i_bIsNumber				:= FALSE);
						
s_fbParamTeslaMeterPort(i_fDefaultValue			:= 0,
						i_nArrayFolderIndex		:= 1,
						i_sName					:= 'Tesla meter port number',
						i_bIsNumber				:= TRUE);

//---------

						
s_fbParamTotalStroke(i_fDefaultValue			:= 100,
						i_nArrayFolderIndex		:= 2,
						i_sName					:= 'Total measurement stroke',
						i_bIsNumber				:= TRUE);
						
s_fbParamStepStroke(i_fDefaultValue				:= 10,
						i_nArrayFolderIndex		:= 2,
						i_sName					:= 'Step distance per measurement',
						i_bIsNumber				:= TRUE);

s_fbParamAveragingNumberTest(i_fDefaultValue		:= 10,
							i_nArrayFolderIndex		:= 2,
							i_sName					:= 'Number of measurements per step for averaging the magnetic field',
							i_bIsNumber				:= TRUE);
							
s_fbParamaMaxMagnitudeCriteria(i_fDefaultValue		:= 100,
							i_nArrayFolderIndex		:= 2,
							i_sName					:= 'Maximum allowed magnitude magnetic field (Test)',
							i_bIsNumber				:= TRUE);

s_fbParamRefIduBottom(i_fDefaultValue				:= 0,
							i_nArrayFolderIndex		:= 2,
							i_sName					:= 'Distance from home position to lower IDU Bottom',
							i_bIsNumber				:= TRUE);
							
s_fbParamRefItm(i_fDefaultValue						:= 0,
							i_nArrayFolderIndex		:= 2,
							i_sName					:= 'Distance from home position Itm lower IDU / upper IDU',
							i_bIsNumber				:= TRUE);
							
s_fbParamRefCenterTpmPipe(i_fDefaultValue			:= 0,
							i_nArrayFolderIndex		:= 2,
							i_sName					:= 'Distance from home position to centre TPM pipe',
							i_bIsNumber				:= TRUE);
							
s_fbParamRefCpValve(i_fDefaultValue		:= 0,
							i_nArrayFolderIndex		:= 2,
							i_sName					:= 'Distance from home position to bottom C/P valve',
							i_bIsNumber				:= TRUE);				

GVL_DataLogging.g_stReportData.CabinetSerialNumber      := s_fbParamToolHardwareNr.p_sValue;
GVL_DataLogging.g_stReportData.TesterSoftwareVersion    := s_fbParamToolSoftwareVersion.p_sValue;
GVL_DataLogging.g_stReportData.Operator                 := GVL.g_sUser;
GVL_DataLogging.g_stReportData.Note						:= GVL.g_sNotesEntry;
//GVL_DataLogging.g_stReportData.Message can be filled in test procedure with for example the error if test is stopped
GVL_DataLogging.g_stReportData.SerialNumber             := GVL.g_sSerialNumber;

s_fToHmiXAxisMin	:= -2*s_fbParamaMaxMagnitudeCriteria.p_fValue;
s_fToHmiXAxisMax	:= 2*s_fbParamaMaxMagnitudeCriteria.p_fValue;
s_fToHmiYAxisMin	:= s_CmProbeMotor.p_fHomePosition;
s_fToHmiYAxisMax	:= s_fbParamRefCpValve.p_fValue*1.2;

_m_Params := TRUE;
END_METHOD

METHOD PRIVATE _m_PrepareDataFile : BOOL
VAR CONSTANT
	c_nStartRow : UINT := 10;
END_VAR
VAR_INPUT
	i_nTotalMeasurementSteps : UINT;
END_VAR
VAR
	t_nCounter : UINT;
END_VAR
//Tester data
GVL_DataLogging.g_aLoggingDataMagnetic[1,2] := GVL_DataLogging.g_stReportData.CabinetSerialNumber;
GVL_DataLogging.g_aLoggingDataMagnetic[2,2] := GVL_DataLogging.g_stReportData.TesterSoftwareVersion;
GVL_DataLogging.g_aLoggingDataMagnetic[3,2] := GVL_DataLogging.g_stReportData.Operator;
GVL_DataLogging.g_aLoggingDataMagnetic[4,2] := GVL_DataLogging.g_stReportData.Message;
GVL_DataLogging.g_aLoggingDataMagnetic[5,2] := GVL_DataLogging.g_stReportData.Note;
GVL_DataLogging.g_aLoggingDataMagnetic[6,2] := GVL_KMWEGenericLib.g_fbCurrentTime.p_sCurrentDateTime_File;
GVL_DataLogging.g_aLoggingDataMagnetic[7,2] := GVL_DataLogging.g_stReportData.SerialNumber;	
GVL_DataLogging.g_aLoggingDataMagnetic[8,2] := s_sTestResult;	

//Product and test data
FOR t_nCounter := 0 TO i_nTotalMeasurementSteps DO
	GVL_DataLogging.g_aLoggingDataMagnetic[c_nStartRow+t_nCounter,1] :=	TO_STRING(s_aProbePositionZ[t_nCounter]);	
	GVL_DataLogging.g_aLoggingDataMagnetic[c_nStartRow+t_nCounter,2] := TO_STRING(s_aMagneticX[t_nCounter]);
	GVL_DataLogging.g_aLoggingDataMagnetic[c_nStartRow+t_nCounter,3] :=	TO_STRING(s_aMagneticY[t_nCounter]);
	GVL_DataLogging.g_aLoggingDataMagnetic[c_nStartRow+t_nCounter,4] :=	TO_STRING(s_aMagneticZ[t_nCounter]);
	GVL_DataLogging.g_aLoggingDataMagnetic[c_nStartRow+t_nCounter,5] :=	TO_STRING(s_aMagneticMagnitude[t_nCounter]);
END_FOR

_m_PrepareDataFile := TRUE;
END_METHOD

METHOD PRIVATE _m_Procedure_Test : E_STATE
VAR_INPUT
	i_bCmdReset			: BOOL;
	i_bStaError			: BOOL;
END_VAR
VAR_INST
	//Sequence control
	s_eSequence				: E_TestProcedure_Steps;
	s_fbSeqControl			: FB_SeqControl;
		
	//Error handling
	s_bErrorDBSaveDone			: BOOL;
	s_bErrorHandlingDone		: BOOL;
	
	//Measurements
	s_nTotalMeasurementSteps 	: UINT;
	s_nMeasurementStep		 	: UINT; 	

	s_fSimulationNumber			: LREAL;
	
	s_sXMLDataRow				: T_MAXSTRING;
	
END_VAR

VAR
	t_nCounterPolish			: UINT;
	t_nCyclceReplies			: UDINT := 1;
END_VAR
s_fbSeqControl(
	i_nSeqStep:= s_eSequence, 
	i_sStepName:= TO_STRING(s_eSequence), 
	i_bCmdReset:= i_bCmdReset, 
	i_bStaError:= i_bStaError,  
	q_eActState=> _m_Procedure_Test);
	
IF _m_Procedure_Test = E_State.Busy THEN
	s_nToHmiStepNr := s_eSequence; 	
	
	s_fbHmiBtnStop.p_bStaEnabled := TRUE;
	s_fbHmiBtnStop.p_bStaVisible := TRUE;		
END_IF									
			
CASE s_eSequence OF
	E_TestProcedure_Steps.Idle:
		;
	
	E_TestProcedure_Steps.Start:
		IF s_fbSeqControl.q_bStaEntry THEN
			MEMSET(ADR(GVL_DataLogging.g_aLoggingDataMagnetic), 0, SIZEOF(GVL_DataLogging.g_aLoggingDataMagnetic));	

			MEMSET(ADR(s_aHmi_MagneticTest)		, 0, SIZEOF(s_aHmi_MagneticTest));
			
			MEMSET(ADR(s_aMagneticX)			, 0, SIZEOF(s_aMagneticX));
			MEMSET(ADR(s_aMagneticY)			, 0, SIZEOF(s_aMagneticY));
			MEMSET(ADR(s_aMagneticZ)			, 0, SIZEOF(s_aMagneticZ));
			MEMSET(ADR(s_aMagneticMagnitude)	, 0, SIZEOF(s_aMagneticMagnitude));
			MEMSET(ADR(s_aProbePositionZ) 		, 0, SIZEOF(s_aProbePositionZ));
		
			MEMSET(ADR(s_sXMLData)				, 0, SIZEOF(s_sXMLData)); 
			
			GVL.g_sToHmiMiddleContent := GVL.g_stHmiMiddle.OperatorPrepareTester;	
			
			s_fbHmiBtnStart.p_bStaEnabled 						:= FALSE;
			s_fbHmiBtnStart.p_bStaVisible 						:= FALSE;
			
			GVL.g_eStaLedColor									:= E_KmweLedColors.Green;
			GVL.g_bLedFlashFast									:= FALSE;
			GVL.g_bLedFlashSlow									:= FALSE;
			
			GVL_KMWEGenericLib.g_fbHmiBtnReturn.p_bStaEnabled	:= FALSE;
			GVL_KMWEGenericLib.g_fbHmiBtnReturn.p_bStaVisible	:= FALSE;

			s_sTestResult				:= 'Busy';
			s_sToHmiProcedure 			:= 'Magnetic field test';
			s_nToHmiMaxStepNr 			:= TO_INT(E_TestProcedure_Steps.OperatorDisconnect);

			s_nTotalMeasurementSteps 	:= TO_UINT(s_fbParamTotalStroke.p_fValue/s_fbParamStepStroke.p_fValue);
			s_nMeasurementStep			:= 0;
			
			s_fSimulationNumber			:= 2;
		END_IF
		
		s_eSequence := E_TestProcedure_Steps.ConnectDb;
		
	E_TestProcedure_Steps.ConnectDb:
		IF s_fbSeqControl.q_bStaEntry THEN
			s_sToHmiInstructionText := 'Connecting to the DB';
		END_IF
			
		IF GVL_Datalogging.g_fbSqlDatabase.m_Connect() 
			AND GVL_KMWEGenericLib.g_fbCurrentTime.m_GetTime() 
		THEN
			s_eSequence := E_TestProcedure_Steps.InitializeDB;
		END_IF

	E_TestProcedure_Steps.InitializeDB:
			IF s_fbSeqcontrol.q_bStaEntry THEN	
				s_sToHmiInstructionText := 'Initialize a new DB entry';
			END_IF
			
			IF GVL_Datalogging.g_fbSqlDatabase.m_NewTableRow(i_sTableName 	:= GVL_Datalogging.c_sTableNameMagnetic,
												i_sIdentificationColumnName := GVL_Datalogging.c_sIdentificationColumnDataTime,
												i_sIdentificationValue		:=	GVL_KMWEGenericLib.g_fbCurrentTime.p_sCurrentDateTime_DB)
			THEN
				s_eSequence := E_TestProcedure_Steps.InitializeDataLogging;
			END_IF
	
	E_TestProcedure_Steps.InitializeDataLogging:
		IF s_fbSeqcontrol.q_bStaEntry THEN	
			s_sToHmiInstructionText := 'Initialize a new result file';
			
			GVL_DataLogging.g_eDataAction		:= E_DataReadWriteActions.MagneticProcedure;
			GVL_DataLogging.g_sFilenameFast		:= 'Data\InitialTest';	
		END_IF
		
		GVL_DataLogging.g_bCmdResetReadFast 		:= s_fbSeqControl.q_bStaEntry;

		IF GVL_DataLogging.g_fbDataLogger.q_eStaReadFast = E_State.Ready 
			AND NOT s_fbSeqControl.q_bStaEntry THEN
			s_eSequence := E_TestProcedure_Steps.OperatorMounting;
		END_IF
				
	E_TestProcedure_Steps.OperatorMounting:
		IF s_fbSeqControl.q_bStaEntry THEN
			s_sToHmiInstructionText 								:= 'Placement of test product';
			
			GVL.g_bLedFlashSlow										:= TRUE;
			GVL_KMWEGenericLib.g_fbHmiBtnAcknowledge.p_bStaVisible	:= TRUE;
		END_IF
		
		GVL_KMWEGenericLib.g_fbHmiBtnAcknowledge.p_bStaEnabled		:= GVL.g_UnRMMT.s_diEmergencyBtn.p_bStaInput OR GVL.g_fbHmiBtnSimulation.p_bStaBtn;
											
		IF GVL_KMWEGenericLib.g_fbHmiBtnAcknowledge.p_osrBtnPress THEN
 			GVL.g_bLedFlashSlow										:= FALSE;
			GVL_KMWEGenericLib.g_fbHmiBtnAcknowledge.p_bStaEnabled	:= FALSE;
			GVL_KMWEGenericLib.g_fbHmiBtnAcknowledge.p_bStaVisible	:= FALSE;
			
			s_CmProbeMotor.i_bReqEnable								:= TRUE;
			s_CmTeslaMeter.i_bReqEnable								:= TRUE;

			GVL.g_sToHmiMiddleContent 								:= GVL.g_stHmiMiddle.OperatorMoveDown;	
			s_eSequence 											:= E_TestProcedure_Steps.OperatorMoveTable;
		END_IF
		
	E_TestProcedure_Steps.OperatorMoveTable:	
		IF s_fbSeqControl.q_bStaEntry THEN
			s_sToHmiInstructionText 								:= 'Placement of test product';
			GVL.g_bConnectTestEquipment								:= TRUE;
			GVL.g_bLedFlashSlow										:= TRUE;
			
			GVL_KMWEGenericLib.g_fbHmiBtnAcknowledge.p_bStaVisible	:= TRUE;
		END_IF
	
		s_doRelayTableDown.i_bStaOutput	:= NOT s_diTableDownSensor.p_bStaInput 
											AND s_diBtnTableDown.p_bStaInput 
											AND NOT s_diBtnStop.p_bStaInput;
	
		GVL_KMWEGenericLib.g_fbHmiBtnAcknowledge.p_bStaEnabled	:= s_diBtnTableDown.p_bStaInput OR GVL.g_fbHmiBtnSimulation.p_bStaBtn;
											
		IF GVL_KMWEGenericLib.g_fbHmiBtnAcknowledge.p_osrBtnPress THEN
			GVL.g_bLedFlashSlow										:= FALSE;
			GVL_KMWEGenericLib.g_fbHmiBtnAcknowledge.p_bStaEnabled	:= FALSE;
			GVL_KMWEGenericLib.g_fbHmiBtnAcknowledge.p_bStaVisible	:= FALSE;
			
			s_CmProbeMotor.i_bReqEnable								:= TRUE;
			s_CmTeslaMeter.i_bReqEnable								:= TRUE;

			GVL.g_sToHmiMiddleContent 	:= GVL.g_stHmiMiddle.ProcedureTesting;	
			s_eSequence 				:= E_TestProcedure_Steps.EnableMotor;
		END_IF	
			
	E_TestProcedure_Steps.EnableMotor:
		IF s_fbSeqcontrol.q_bStaEntry THEN
			s_sToHmiInstructionText := 'Enabling probe motor';	
		END_IF
		
		IF s_CmProbeMotor.m_EnableAxis() THEN
			s_eSequence 	:= E_TestProcedure_Steps.HomeMotor;
		END_IF
		
	E_TestProcedure_Steps.HomeMotor:
		IF s_fbSeqControl.q_bStaEntry THEN
			s_sToHmiInstructionText := 'Motor homing';	
		END_IF
		
		IF NOT GVL.g_fbHmiBtnSimulation.p_bStaBtn THEN
			IF s_CmProbeMotor.m_HomeMotor() THEN
				s_eSequence := E_TestProcedure_Steps.MoveToStart;
			END_IF
		ELSE
			IF s_CmProbeMotor.m_SetPosition(i_fPosition := 0) THEN
				s_eSequence := E_TestProcedure_Steps.MoveToStart;
			END_IF
		END_IF
		
	E_TestProcedure_Steps.MoveToStart:
		IF s_fbSeqControl.q_bStaEntry THEN
			s_sToHmiInstructionText := 'Moving to start position';	
		END_IF	
		
		IF s_CmProbeMotor.m_MoveAbsolute(i_fSetPosition := 0) THEN
			s_eSequence := E_TestProcedure_Steps.DisableMotor;
		END_IF

		
	E_TestProcedure_Steps.DisableMotor:
		IF s_fbSeqcontrol.q_bStaEntry THEN
			s_sToHmiInstructionText := 'Disable probe motor before measurement';	
		END_IF
	
		IF s_CmProbeMotor.m_DisableAxis() THEN
			IF NOT GVL.g_fbHmiBtnSimulation.p_bStaBtn THEN
				s_eSequence 	:= E_TestProcedure_Steps.ConnectTesla;
			ELSE
				s_eSequence 	:= E_TestProcedure_Steps.CalculateData;
			END_IF
		END_IF

	E_TestProcedure_Steps.ConnectTesla:
		IF s_fbSeqcontrol.q_bStaEntry THEN
			s_sToHmiInstructionText := 'Connecting to probe';	
			
			s_CmTeslaMeter.i_stSettings.sMetrelIpAdress := s_fbParamTeslaMeterIp.p_sValue;
			s_CmTeslaMeter.i_stSettings.sMetrelPort 	:= TO_UDINT(s_fbParamTeslaMeterPort.p_fValue);

		END_IF
		
		IF GVL.g_fbHmiBtnSimulation.p_bStaBtn THEN
			s_eSequence 	:= E_TestProcedure_Steps.CalculateData;
		ELSIF  s_CmTeslaMeter.m_Connect() THEN
			s_eSequence 	:= E_TestProcedure_Steps.ConfigureTesla;
		END_IF
		
	E_TestProcedure_Steps.ConfigureTesla:
		IF s_fbSeqcontrol.q_bStaEntry THEN
			s_sToHmiInstructionText := 'Configuring to probe';	
		END_IF
		
		IF s_CmTeslaMeter.m_SendCommand(i_sCommand := s_stCommandsTesla.sSetModeDC , i_bAddCRChar := FALSE) THEN
			s_eSequence 	:= E_TestProcedure_Steps.MeasureMagneticField;
		END_IF

	E_TestProcedure_Steps.MeasureMagneticField:
		IF s_fbSeqcontrol.q_bStaEntry THEN
			s_sToHmiInstructionText := CONCAT('Measure magnetic field, ',
										 	CONCAT('Measurement: ', 
											CONCAT(TO_STRING(s_nMeasurementStep),
											CONCAT('/',TO_STRING(s_nTotalMeasurementSteps)))));
		
		END_IF
		
		IF _m_GetMagneticField(i_bCmdReset 		:= s_fbSeqControl.q_bStaEntry,
								q_fMagneticX 	=> s_aMagneticX[s_nMeasurementStep],
								q_fMagneticY 	=> s_aMagneticY[s_nMeasurementStep],
								q_fMagneticZ 	=> s_aMagneticZ[s_nMeasurementStep]) = E_STATE.Ready 
		THEN
			s_eSequence := 	E_TestProcedure_Steps.CalculateData;
		END_IF
		
	E_TestProcedure_Steps.CalculateData:
		IF s_fbSeqControl.q_bStaEntry THEN
			s_sToHmiInstructionText := CONCAT('Calculate magnetic field, ',
										 	CONCAT('Measurement: ', 
											CONCAT(TO_STRING(s_nMeasurementStep),
											CONCAT('/',TO_STRING(s_nTotalMeasurementSteps)))));	
		
			s_aProbePositionZ[s_nMeasurementStep] 		:= s_CmProbeMotor.p_fActualPos;
			
			IF GVL.g_fbHmiBtnSimulation.p_bStaBtn THEN		
				s_aMagneticX[s_nMeasurementStep] 			:= 10*s_fSimulationNumber+ s_fSimulationNumber;
				s_aMagneticY[s_nMeasurementStep] 			:= -5*s_fSimulationNumber - 3*s_fSimulationNumber/222;
				s_aMagneticZ[s_nMeasurementStep] 			:= -12.0*s_fSimulationNumber + 0.3*s_fSimulationNumber*s_fSimulationNumber;
				s_aMagneticMagnitude[s_nMeasurementStep]	:= SQRT((s_aMagneticX[s_nMeasurementStep]*s_aMagneticX[s_nMeasurementStep]) + (s_aMagneticY[s_nMeasurementStep] * s_aMagneticY[s_nMeasurementStep]));
				s_fSimulationNumber 						:= s_fSimulationNumber + 1;
			ELSE  
				s_aMagneticMagnitude[s_nMeasurementStep]	:= SQRT((s_aMagneticX[s_nMeasurementStep]*s_aMagneticX[s_nMeasurementStep]) + (s_aMagneticY[s_nMeasurementStep] * s_aMagneticY[s_nMeasurementStep]));
			END_IF
						
			//HMI plotting
			s_aHmi_MagneticTest[1,s_nMeasurementStep].x	:= s_aMagneticX[s_nMeasurementStep];
			s_aHmi_MagneticTest[2,s_nMeasurementStep].x := s_aMagneticY[s_nMeasurementStep];
			s_aHmi_MagneticTest[3,s_nMeasurementStep].x := s_aMagneticMagnitude[s_nMeasurementStep];
 
			
			s_aHmi_MagneticTest[1,s_nMeasurementStep].y := s_aProbePositionZ[s_nMeasurementStep];
			s_aHmi_MagneticTest[2,s_nMeasurementStep].y := s_aProbePositionZ[s_nMeasurementStep];
			s_aHmi_MagneticTest[3,s_nMeasurementStep].y := s_aProbePositionZ[s_nMeasurementStep];

			
			FOR t_nCounterPolish := s_nMeasurementStep+1 TO c_nResultDataSize DO
				IF s_nMeasurementStep > 0 THEN
					s_aHmi_MagneticTest[1,t_nCounterPolish].x 			:= s_aHmi_MagneticTest[1,s_nMeasurementStep-1].x;
					s_aHmi_MagneticTest[2,t_nCounterPolish].x 			:= s_aHmi_MagneticTest[2,s_nMeasurementStep-1].x;
					s_aHmi_MagneticTest[3,t_nCounterPolish].x 			:= s_aHmi_MagneticTest[3,s_nMeasurementStep-1].x;

					s_aHmi_MagneticTest[1,t_nCounterPolish].y			:= s_aHmi_MagneticTest[1,s_nMeasurementStep-1].y;
					s_aHmi_MagneticTest[2,t_nCounterPolish].y			:= s_aHmi_MagneticTest[2,s_nMeasurementStep-1].y;
					s_aHmi_MagneticTest[3,t_nCounterPolish].y			:= s_aHmi_MagneticTest[3,s_nMeasurementStep-1].y;
				END_IF
			END_FOR
		END_IF
		
		//Data handling DB
		s_sXMLDataRow := '' ;
		
		s_sXMLDataRow := CONCAT(s_sXMLDataRow, '<row>');
		s_sXMLDataRow := CONCAT(s_sXMLDataRow, 
								CONCAT('<Height>', 
								CONCAT(LREAL_TO_FMTSTR(s_aProbePositionZ[s_nMeasurementStep], 2, TRUE ), '</Height>')));  // Assuming Height is in column 1
		s_sXMLDataRow := CONCAT(s_sXMLDataRow, 
							CONCAT('<Bx>', 
							CONCAT(LREAL_TO_FMTSTR(s_aMagneticX[s_nMeasurementStep], 2, TRUE ), '</Bx>')));  // Assuming Bx is in column 2
		s_sXMLDataRow := CONCAT(s_sXMLDataRow, 
							CONCAT('<By>', 
							CONCAT(LREAL_TO_FMTSTR(s_aMagneticY[s_nMeasurementStep], 2, TRUE ), '</By>')));  // Assuming By is in column 3
		s_sXMLDataRow := CONCAT(s_sXMLDataRow, 
							CONCAT('<Bz>', 
							CONCAT(LREAL_TO_FMTSTR(s_aMagneticZ[s_nMeasurementStep], 2, TRUE ), '</Bz>')));  // Assuming Bz is in column 4
		s_sXMLDataRow := CONCAT(s_sXMLDataRow, 
							CONCAT('<BxyTotal>', 
							CONCAT(LREAL_TO_FMTSTR(s_aMagneticMagnitude[s_nMeasurementStep], 2, TRUE ), '</BxyTotal>')));  // Assuming BxyTotal is in column 5
		s_sXMLDataRow := CONCAT(s_sXMLDataRow, '</row>');
	
		CONCAT2(ADR(s_sXMLData), ADR(s_sXMLDataRow), ADR(s_sXMLData), SIZEOF(s_sXMLData));
		
		//Check if test is finished
		IF s_nMeasurementStep = s_nTotalMeasurementSteps THEN
			s_eSequence := E_TestProcedure_Steps.PassFail;
		ELSE
			s_eSequence := E_TestProcedure_Steps.EnableMotorMeasuring;
		END_IF	
			
	E_TestProcedure_Steps.EnableMotorMeasuring:
		IF s_fbSeqcontrol.q_bStaEntry THEN
			s_sToHmiInstructionText := CONCAT('Enabling probe motor',
										 	CONCAT('Measurement: ', 
											CONCAT(TO_STRING(s_nMeasurementStep),
											CONCAT('/',TO_STRING(s_nTotalMeasurementSteps)))));	
		END_IF
		
		IF s_CmProbeMotor.m_EnableAxis() THEN
			s_eSequence 	:= E_TestProcedure_Steps.MoveMotorToNextPos;
		END_IF	
		
	E_TestProcedure_Steps.MoveMotorToNextPos:
		IF s_fbSeqcontrol.q_bStaEntry THEN
			s_nMeasurementStep		:= s_nMeasurementStep + 1;
			s_sToHmiInstructionText := CONCAT('Moving to next position, ',
										 	CONCAT('Measurement: ', 
											CONCAT(TO_STRING(s_nMeasurementStep),
											CONCAT('/',TO_STRING(s_nTotalMeasurementSteps)))));	
		END_IF
		
		IF s_CmProbeMotor.m_MoveAbsolute(i_fSetPosition := s_fbParamStepStroke.p_fValue * s_nMeasurementStep) THEN
			s_eSequence := E_TestProcedure_Steps.DisableMotorMeasuring;
		END_IF	
		
	E_TestProcedure_Steps.DisableMotorMeasuring:
		IF s_fbSeqcontrol.q_bStaEntry THEN	
			s_sToHmiInstructionText := CONCAT('Disabling probe motor, ',
										 	CONCAT('Measurement: ', 
											CONCAT(TO_STRING(s_nMeasurementStep),
											CONCAT('/',TO_STRING(s_nTotalMeasurementSteps)))));		
		END_IF
		
		IF s_CmProbeMotor.m_DisableAxis() THEN
			IF NOT GVL.g_fbHmiBtnSimulation.p_bStaBtn THEN
				s_eSequence 	:= E_TestProcedure_Steps.MeasureMagneticField;
			ELSE
				s_eSequence 	:= E_TestProcedure_Steps.CalculateData;
			END_IF
		END_IF	
		
	E_TestProcedure_Steps.PassFail:
		s_sToHmiInstructionText := 'Pass fail';

		FOR t_nCounterPolish := 0 TO c_nResultDataSize DO
			IF s_aMagneticMagnitude[t_nCounterPolish] > s_fbParamaMaxMagnitudeCriteria.p_fValue  
			THEN
				s_sTestResult 		:= 'Fail';
				GVL.g_eStaLedColor 	:= E_KmweLedColors.Red;
				EXIT;
			ELSIF t_nCounterPolish = c_nResultDataSize THEN
				s_sTestResult 		:= 'Pass';
				GVL.g_eStaLedColor 	:= E_KmweLedColors.Green;
			END_IF
		END_FOR
	
		s_eSequence := E_TestProcedure_Steps.DisconnectTesla;
		
	E_TestProcedure_Steps.DisconnectTesla:
		IF s_fbSeqcontrol.q_bStaEntry THEN
			s_sToHmiInstructionText := 'Disconnect to probe';	
		END_IF
		
		IF s_CmTeslaMeter.m_Disconnect() THEN
			s_eSequence 	:= E_TestProcedure_Steps.EnableMotorEnd;
		END_IF
			
	E_TestProcedure_Steps.EnableMotorEnd:
		IF s_fbSeqcontrol.q_bStaEntry THEN
			s_sToHmiInstructionText := 'Enabling probe motor';	
		END_IF
		
		IF s_CmProbeMotor.m_EnableAxis() THEN
			s_eSequence 	:= E_TestProcedure_Steps.MoveMotorEnd;
		END_IF	
		
	E_TestProcedure_Steps.MoveMotorEnd:
		IF s_fbSeqcontrol.q_bStaEntry THEN
			s_sToHmiInstructionText := 'Moving end position';
		END_IF
		
		IF s_CmProbeMotor.m_MoveAbsolute(i_fSetPosition := s_CmProbeMotor.p_fHomePosition) THEN
			s_eSequence := E_TestProcedure_Steps.DisableMotorEnd;
		END_IF	
		
	E_TestProcedure_Steps.DisableMotorEnd:
		IF s_fbSeqcontrol.q_bStaEntry THEN
			s_sToHmiInstructionText := 'Disabling probe motor end';	
		END_IF
		
		IF s_CmProbeMotor.m_DisableAxis() THEN
			s_eSequence 	:= E_TestProcedure_Steps.WriteDataDb;
		END_IF

	E_TestProcedure_Steps.WriteDataDb:
		IF s_fbSeqControl.q_bStaEntry THEN	
			s_sToHmiInstructionText 	:= 'Logging data to DB';	
		END_IF

		IF  _m_DatabaseMagnetic(i_bCmdReset				:= s_fbSeqControl.q_bStaEntry,
									i_sPassFail				:= s_sTestResult) 
		THEN
			s_eSequence := E_TestProcedure_Steps.DisconnectDb;
		END_IF	
		
	E_TestProcedure_Steps.DisconnectDb:
		s_sToHmiInstructionText := 'Disconnect DB';
		
		IF GVL_Datalogging.g_fbSqlDatabase.m_Disconnect() THEN
			s_eSequence := E_TestProcedure_Steps.WriteDataLogging;
		END_IF
					
	E_TestProcedure_Steps.WriteDataLogging:
		IF s_fbSeqControl.q_bStaEntry THEN	
			s_sToHmiInstructionText 			:= 'Logging data';	
			GVL_Datalogging.g_bStartDataLogger  := TRUE;
			GVL_KMWEGenericLib.g_fbCurrentTime.m_GetTime();

			_m_PrepareDataFile(i_nTotalMeasurementSteps := s_nTotalMeasurementSteps);
			
			GVL_DataLogging.g_sFilenameFast := CONCAT('Data\T_', 
												CONCAT(GVL_DataLogging.g_stReportData.SerialNumber, 
												CONCAT('_', 
												CONCAT(GVL_DataLogging.g_stReportData.Operator, 
												CONCAT('_', GVL_KMWEGenericLib.g_fbCurrentTime.p_sCurrentDateTime_File)))));

			GVL_DataLogging.g_eDataAction	:= E_DataReadWriteActions.MagneticProcedure;
		ELSE
			GVL_DataLogging.g_bCmdResetWriteFast 	:= GVL_DATALOGGING.g_bStartDataLogger;
	
			IF GVL_DataLogging.g_fbDataLogger.q_eStaWriteFast = E_State.Ready 
				AND NOT GVL_Datalogging.g_bStartDataLogger
			THEN
				GVL.g_bLedFlashSlow										:= TRUE;
				GVL.g_osrNotify.CLK										:= TRUE;	
				GVL_KMWEGenericLib.g_fbHmiBtnAcknowledge.p_bStaEnabled	:= TRUE;
				GVL_KMWEGenericLib.g_fbHmiBtnAcknowledge.p_bStaVisible	:= TRUE;
				
				IF GVL_KMWEGenericLib.g_fbHmiBtnAcknowledge.p_osrBtnPress THEN
					s_eSequence := E_TestProcedure_Steps.OperatorDisconnect;
				END_IF
			END_IF
			
			GVL_Datalogging.g_bStartDataLogger  := FALSE;
		END_IF
		
	E_TestProcedure_Steps.OperatorDisconnect:
		IF s_fbSeqControl.q_bStaEntry THEN	
			s_sToHmiInstructionText 		:= 'Removal of test product';	
			
			s_CmProbeMotor.i_bReqEnable		:= FALSE;
			s_CmTeslaMeter.i_bReqEnable		:= FALSE;
			GVL.g_bConnectTestEquipment		:= FALSE;
			GVL.g_sToHmiMiddleContent		:= GVL.g_stHmiMiddle.OperatorDisconnect;
			
			GVL_KMWEGenericLib.g_fbHmiBtnAcknowledge.p_bStaVisible 	:= TRUE;
		END_IF
		
		GVL_KMWEGenericLib.g_fbHmiBtnAcknowledge.p_bStaEnabled		:= NOT GVL.g_UnRMMT.s_diEmergencyBtn.p_bStaInput OR GVL.g_fbHmiBtnSimulation.p_bStaBtn;
											
		IF GVL_KMWEGenericLib.g_fbHmiBtnAcknowledge.p_osrBtnPress THEN
 			GVL.g_bLedFlashSlow										:= FALSE;
			GVL_KMWEGenericLib.g_fbHmiBtnAcknowledge.p_bStaEnabled	:= FALSE;
			GVL_KMWEGenericLib.g_fbHmiBtnAcknowledge.p_bStaVisible	:= FALSE;
			
			s_eSequence 											:= E_TestProcedure_Steps.Ready;
		END_IF

	E_TestProcedure_Steps.Ready:
		IF s_fbSeqControl.q_bStaEntry THEN	
			s_sToHmiInstructionText 	:= 'Done';	
			
			s_CmProbeMotor.i_bReqEnable								:= FALSE;
			s_CmTeslaMeter.i_bReqEnable								:= FALSE;
		
			GVL_KMWEGenericLib.g_fbHmiBtnReturn.p_bStaVisible 		:= FALSE;
			GVL_KMWEGenericLib.g_fbHmiBtnReturn.p_bStaEnabled 		:= FALSE;
			
			GVL.g_UnRMMT.p_eCtrlMode := E_CtrlMode.IDLE;
			
			GVL_KMWEGenericLib.g_fbParamManager.p_bShowHmiParam := FALSE;

			GVL.g_sToHmiMiddleContent 	:= GVL.g_stHmiMiddle.Start;
			GVL.g_sToHmiBottomContent	:= GVL.g_stHmiBottomBar.Start;
		END_IF
		
	E_TestProcedure_Steps.Error:
		IF s_fbSeqControl.q_bStaEntry THEN
			s_sToHmiInstructionText :=  'ERROR: Process interupted';
			
			GVL.g_bLedFlashSlow		:= FALSE;
			GVL.g_bLedFlashFast		:= TRUE;
			
			s_bErrorDBSaveDone			:= FALSE;
			s_bErrorHandlingDone		:= FALSE;
				
			GVL.g_sToHmiBottomContent 	:= GVL.g_stHmiBottomBar.General_ReturnToStart;
			
			GVL_KMWEGenericLib.g_fbHmiBtnReturnToStart.p_bStaVisible 		:= FALSE;
			GVL_KMWEGenericLib.g_fbHmiBtnReturnToStart.p_bStaEnabled 		:= FALSE;
			
			GVL_KMWEGenericLib.g_fbHmiBtnReturn.p_bStaVisible 				:= FALSE;
			GVL_KMWEGenericLib.g_fbHmiBtnReturn.p_bStaEnabled 				:= FALSE;	
			
			GVL_KMWEGenericLib.g_fbHmiBtnAcknowledge.p_bStaVisible			:= FALSE;
			GVL_KMWEGenericLib.g_fbHmiBtnAcknowledge.p_bStaEnabled			:= FALSE;
		END_IF
	
		IF s_CmTeslaMeter.p_bConnected THEN
			s_CmTeslaMeter.m_Disconnect();
		END_IF
		
		IF s_CmProbeMotor.p_bStaMoving THEN
			s_CmProbeMotor.m_StopMoving();
		END_IF
		
		IF NOT s_CmProbeMotor.p_bStaMoving 
			AND s_CmProbeMotor.p_bStaEnabled
		THEN
			s_CmProbeMotor.m_DisableAxis();
		END_IF
		
		IF NOT GVL_Datalogging.g_fbSqlDatabase.p_bStaError 
			AND GVL_Datalogging.g_fbSqlDatabase.p_bStaConnected  
			AND NOT s_bErrorDBSaveDone
		THEN
			IF _m_DatabaseMagnetic(i_bCmdReset				:= s_fbSeqControl.q_bStaEntry,
									i_sPassFail				:= s_sTestResult) 
			THEN
				s_bErrorDbSaveDone := TRUE;
			END_IF
		END_IF
		
		IF s_bErrorDbSaveDone AND NOT s_bErrorHandlingDone THEN
			IF GVL_Datalogging.g_fbSqlDatabase.m_Disconnect() THEN
				s_bErrorHandlingDone := TRUE;
			END_IF
		END_IF
		
		IF NOT s_CmProbeMotor.p_bStaEnabled AND NOT s_CmTeslaMeter.p_bConnected THEN
			IF s_bErrorHandlingDone THEN
				s_sToHmiInstructionText :=  'ERROR: start test again';
			ELSE
				s_sToHmiInstructionText :=  'ERROR: start test again (Db error so no data saved)';
			END_IF
			
			s_CmProbeMotor.i_bReqEnable									:= FALSE;
			s_CmTeslaMeter.i_bReqEnable									:= FALSE;
	
			GVL_KMWEGenericLib.g_fbHmiBtnReturnToStart.p_bStaVisible 	:= TRUE;
			GVL_KMWEGenericLib.g_fbHmiBtnReturnToStart.p_bStaEnabled 	:= TRUE;

			IF (GVL_KMWEGenericLib.g_fbHmiBtnReturn.p_osrBtnPress AND GVL.g_sToHmiMiddleContent <> GVL.g_stHmiMiddle.AlarmManager)
			 OR GVL_KMWEGenericLib.g_fbHmiBtnReturnToStart.p_osrBtnPress  THEN
				s_eCurrentTest 											:= E_TestMode.IDLE;
				
				GVL_KMWEGenericLib.g_fbHmiBtnReturnToStart.p_bStaVisible 	:= FALSE;
				GVL_KMWEGenericLib.g_fbHmiBtnReturnToStart.p_bStaEnabled 	:= FALSE;
	
				GVL.g_sToHmiMiddleContent 	:= GVL.g_stHmiMiddle.Start;
			END_IF
		END_IF		
END_CASE
END_METHOD

METHOD PUBLIC m_Main : BOOL
IF NOT SUPER^.m_Main() THEN
	RETURN;
END_IF

CASE i_eCtrlMode OF
	E_CtrlMode.IDLE:
		IF s_CmProbeMotor.p_bStaEnabled THEN
			s_CmProbeMotor.m_DisableAxis();
			s_fbHmiBtnEnableMotor.m_Off();
			s_fbHmiBtnHomeMotor.p_bStaEnabled := FALSE;
		END_IF
		
		s_eCurrentTest	:= 	E_TestMode.IDLE;
	
		s_fbHmiBtnStop.p_bStaVisible := FALSE;
		s_fbHmiBtnStop.p_bStaEnabled := FALSE;		
		
	E_CtrlMode.AUTOMATIC:
		
		CASE s_eCurrentTest OF
			E_TestMode.IDLE:
				GVL.g_bLedFlashSlow			:= FALSE;
				
				s_CmProbeMotor.i_bReqEnable	:= FALSE;
			
				GVL_KMWEGenericLib.g_fbHmiBtnReturn.p_bStaEnabled 	:= TRUE;
				GVL_KMWEGenericLib.g_fbHmiBtnReturn.p_bStaVisible 	:= TRUE;
				
				IF GVL.g_sToHmiMiddleContent = GVL.g_stHmiMiddle.OperatorInputData THEN
					IF NOT GVL_KMWEGenericLib.g_fbAlarmManager.p_bAlarmActive THEN
						s_fbHmiBtnStart.p_bStaVisible	:= TRUE;
						s_fbHmiBtnStart.p_bStaEnabled	:= TRUE;
					ELSE
						s_fbHmiBtnStart.p_bStaVisible	:= FALSE;
						s_fbHmiBtnStart.p_bStaEnabled	:= FALSE;
					END_IF
				END_IF
				
				IF s_fbHmiBtnStart.p_osrBtnPress THEN
					s_eCurrentTest := E_TestMode.Magnetic; 
				END_IF 
				
			E_TestMode.Magnetic:	
				_m_Procedure_Test(i_bCmdReset			:= s_fbHmiBtnStart.p_osfBtnPress, 
									i_bStaError			:= GVL_KMWEGenericLib.g_fbAlarmManager.p_bAlarmActive OR s_fbHmiBtnStop.p_osrBtnPress OR s_diBtnStop.p_osrOn);
		END_CASE
		
	E_CtrlMode.MANUAL:
		_m_Manual(i_bCmdReset			:= GVL.g_UnRMMT.s_fbHmiBtnManual.p_osfBtnPress OR GVL_KMWEGenericLib.g_fbAlarmManager.p_osrReset, 
					i_bStaError			:= GVL_KMWEGenericLib.g_fbAlarmManager.p_bAlarmActive OR s_fbHmiBtnStop.p_osrBtnPress OR s_diBtnStop.p_osrOn);	
END_CASE
END_METHOD

END_FUNCTION_BLOCK

(* stored: Version 1.1.0.1, ProductVersion 3.1.4024.12
   POU EM_Doors: Id {0ea26ddd-052a-4260-bfaf-0daade60103a}, SpecialFunc None
   Folder Administrative: Id {a0739789-5416-422a-bb91-d278e4d6c0c6}
   Folder General: Id {abe66412-5cb4-4e94-938b-00932105d43b}
   Folder Procedures: Id {4fbebc8d-2e5e-4843-ba3a-d70401e17a8b}
   Folder Sensors: Id {b84b418c-1139-4453-87ba-182257d5dca9}
   Method _m_Alarms: Id {34703853-800b-4320-8e6c-49abce8785b7}
   Method _m_DatabaseMagnetic: Id {bb78cd83-18a1-4e68-a34c-6c165cb86cbd}
   Method _m_Devices: Id {c18c3403-a619-4da8-8c16-d38b3f2bd5db}
   Method _m_GetMagneticField: Id {d945ccf2-8199-4155-868a-7f8c730d83f6}
   Method _m_Hmi: Id {06e9697b-07d7-4e29-8455-791381b5d99d}
   Method _m_HmiPlots: Id {cbe7055f-d035-4d00-9575-2b87f9463135}
   Method _m_HmiPlots_Test: Id {ac4d79a0-338a-4f01-97b6-48154040c275}
   Method _m_Init: Id {f5588ebd-495a-4c31-a7f5-23415377d40e}
   Method _m_Inputs: Id {08e3676c-19d2-4657-8762-4d7303d85c82}
   Method _m_Manual: Id {b1ba78d1-de13-4a0c-aa03-999980f6a4be}
   Method _m_Outputs: Id {f763b42e-2a14-49e4-aeec-3b4dc606af2b}
   Method _m_Params: Id {02936153-be53-403e-812d-8d9a77c13756}
   Method _m_PrepareDataFile: Id {fb1741c7-802f-41e2-a9c9-3469959c243c}
   Method _m_Procedure_Test: Id {20c92f11-c293-4bd9-8121-fced590a54bd}
   Method m_Main: Id {c1559ad6-cc3e-4059-9eff-299ddfbeac7b} *)
